(* IEC 61131-3 sources: Mini-Conveyors-Automation/plc, 10 files *)

(* ---- types.st ---- *)
(* =============================================================================
   types.st - Type Definitions
   Mini-Fulfillment Conveyor System

   Enumerations and structures used throughout the PLC program.
   ============================================================================= *)

(* System operating states *)
TYPE E_SystemState :
(
    STOPPED  := 0,   (* System is idle, motor off, safe to interact *)
    STARTING := 1,   (* Pre-run checks in progress *)
    RUNNING  := 2,   (* Normal operation, conveyor moving *)
    FAULT    := 3    (* Fault condition active, motor off, alarm on *)
);
END_TYPE

(* Fault codes *)
TYPE E_FaultCode :
(
    NONE            := 0,   (* No fault *)
    ESTOP           := 1,   (* Emergency stop activated *)
    JAM_INFEED      := 2,   (* Jam detected at infeed photoeye *)
    JAM_DIVERTER    := 3,   (* Jam detected at diverter photoeye *)
    JAM_OUTFEED_B   := 4,   (* Jam detected at outfeed B photoeye *)
    JAM_OUTFEED_C   := 5    (* Jam detected at outfeed C photoeye *)
);
END_TYPE

(* Operating mode *)
TYPE E_OperatingMode :
(
    AUTO   := 0,   (* Automatic mode - full autonomous operation *)
    MANUAL := 1    (* Manual mode - jog only, no auto routing *)
);
END_TYPE

(* Metrics data structure *)
TYPE ST_Metrics :
STRUCT
    diBoxCount       : DINT;    (* Total boxes processed *)
    rAvgCycleTime    : REAL;    (* Average cycle time in seconds *)
    diJamCount       : DINT;    (* Total jam events *)
    rThroughput      : REAL;    (* Current throughput in boxes/hour *)
    rRunningTime     : REAL;    (* Total running time in seconds *)
    rFaultTime       : REAL;    (* Total fault/downtime in seconds *)
    rLastCycleTime   : REAL;    (* Most recent box cycle time *)
    rCycleTimeSum    : REAL;    (* Sum of all cycle times for averaging *)
END_STRUCT
END_TYPE

(* Jam detection status per photoeye *)
TYPE ST_JamStatus :
STRUCT
    bBlocked         : BOOL;    (* Photoeye currently blocked *)
    bJamDetected     : BOOL;    (* Jam threshold exceeded *)
    tBlockedDuration : TIME;    (* How long PE has been blocked *)
END_STRUCT
END_TYPE

(* ---- global_vars.st ---- *)
(* =============================================================================
   global_vars.st - Global Variables (Global Variable List)
   Mini-Fulfillment Conveyor System

   Shared variables used across program blocks and for HMI binding.
   ============================================================================= *)

VAR_GLOBAL
    (* =========================================================================
       SYSTEM STATE
       ========================================================================= *)
    eSystemState    : E_SystemState := STOPPED;    (* Current system state *)
    eOperatingMode  : E_OperatingMode := AUTO;     (* Current operating mode *)
    eFaultCode      : E_FaultCode := NONE;         (* Active fault code *)
    sFaultMessage   : STRING(80) := '';             (* Active fault description *)

    (* =========================================================================
       SAFETY FLAGS
       ========================================================================= *)
    bSafeToRun      : BOOL := FALSE;   (* TRUE when all safety checks pass *)
    bFaultActive    : BOOL := FALSE;   (* TRUE when any fault is active *)
    bEStopLatched   : BOOL := FALSE;   (* TRUE when E-Stop has been activated, requires clear *)
    bJamDetected    : BOOL := FALSE;   (* TRUE when any photoeye jam is detected *)

    (* =========================================================================
       CONTROL FLAGS
       ========================================================================= *)
    bMotorRunCmd    : BOOL := FALSE;   (* Motor run command from state machine *)
    bRejectNext     : BOOL := FALSE;   (* TRUE = next box routes to Station C *)
    diBoxCounter    : DINT := 0;       (* Running box count for routing pattern *)

    (* =========================================================================
       JAM DETECTION STATUS
       ========================================================================= *)
    stJamInfeed     : ST_JamStatus;    (* Jam status for infeed PE *)
    stJamDiverter   : ST_JamStatus;    (* Jam status for diverter PE *)
    stJamOutfeedB   : ST_JamStatus;    (* Jam status for outfeed B PE *)
    stJamOutfeedC   : ST_JamStatus;    (* Jam status for outfeed C PE *)

    (* =========================================================================
       METRICS
       ========================================================================= *)
    stMetrics       : ST_Metrics;      (* Aggregated metrics structure *)

    (* =========================================================================
       HMI INTERFACE - Commands (HMI -> PLC)
       ========================================================================= *)
    bHMI_Start      : BOOL := FALSE;   (* Start command from HMI *)
    bHMI_Stop       : BOOL := FALSE;   (* Stop command from HMI *)
    bHMI_FaultClear : BOOL := FALSE;   (* Fault clear command from HMI *)
    bHMI_JogFwd     : BOOL := FALSE;   (* Jog forward command from HMI (manual mode) *)

    (* =========================================================================
       HMI INTERFACE - Parameters (HMI -> PLC)
       ========================================================================= *)
    rJamTimeoutSec  : REAL := 4.0;     (* Jam detection timeout in seconds (adjustable) *)
    rConveyorSpeed  : REAL := 1.0;     (* Conveyor speed setpoint 0.0 to 1.0 (1.0 = full speed) *)

    (* =========================================================================
       HMI INTERFACE - Status (PLC -> HMI)
       ========================================================================= *)
    iHMI_State      : INT := 0;        (* System state as INT for HMI display *)
    sHMI_FaultMsg   : STRING(80) := '';(* Fault message for HMI display *)
    rHMI_BoxCount   : DINT := 0;       (* Box count for HMI display *)
    rHMI_AvgCycleTime : REAL := 0.0;   (* Avg cycle time for HMI display *)
    rHMI_JamCount   : DINT := 0;       (* Jam count for HMI display *)
    rHMI_Throughput : REAL := 0.0;     (* Throughput for HMI display *)

    (* =========================================================================
       TIMING
       ========================================================================= *)
    tCycleStartTime : TIME := T#0S;    (* Timestamp when current box entered infeed *)
    bCycleActive    : BOOL := FALSE;   (* TRUE when a box is being tracked through the system *)
END_VAR

(* ---- io_mapping.st ---- *)
(* =============================================================================
   io_mapping.st - I/O Address Mapping (Global Variable List)
   Mini-Fulfillment Conveyor System

   Maps physical I/O addresses to symbolic names.
   This GVL is the ONLY place where physical addresses appear.
   All other program blocks reference these symbolic names.
   ============================================================================= *)

VAR_GLOBAL
    (* =========================================================================
       DIGITAL INPUTS
       ========================================================================= *)

    (* Operator panel *)
    bStartPB       AT %IX0.0 : BOOL;   (* Start pushbutton - NO, TRUE on press *)
    bStopPB        AT %IX0.1 : BOOL;   (* Stop pushbutton - NC, FALSE on press *)
    bEStop         AT %IX0.2 : BOOL;   (* E-Stop - NC, FALSE when activated *)
    bModeSelector  AT %IX0.3 : BOOL;   (* Mode switch - FALSE=Auto, TRUE=Manual *)

    (* Photoeyes - TRUE when blocked by a box *)
    bInfeedPE      AT %IX1.0 : BOOL;   (* Infeed photoeye at Station A *)
    bDiverterPE    AT %IX1.1 : BOOL;   (* Diverter photoeye at routing point *)
    bOutfeedBPE    AT %IX1.2 : BOOL;   (* Outfeed B photoeye at Station B (accept) *)
    bOutfeedCPE    AT %IX1.3 : BOOL;   (* Outfeed C photoeye at Station C (reject) *)

    (* =========================================================================
       DIGITAL OUTPUTS
       ========================================================================= *)

    bConveyorMotor     AT %QX0.0 : BOOL;   (* Main conveyor belt motor *)
    bDiverterActuator  AT %QX0.1 : BOOL;   (* Diverter gate solenoid - FALSE=StationB, TRUE=StationC *)
    bAlarmBuzzer       AT %QX0.2 : BOOL;   (* Fault alarm buzzer *)
    bStatusGreen       AT %QX0.3 : BOOL;   (* Green status light - RUNNING *)
    bStatusRed         AT %QX0.4 : BOOL;   (* Red status light - FAULT *)
END_VAR

(* ---- fb_conveyor.st ---- *)
(* =============================================================================
   FB_Conveyor - Conveyor Motor Control Function Block
   Mini-Fulfillment Conveyor System

   Controls the main conveyor belt motor based on system state and mode.
   Provides speed reference output for potential variable-speed drive.
   ============================================================================= *)

FUNCTION_BLOCK FB_Conveyor
VAR_INPUT
    bRunCommand     : BOOL;         (* Motor run command from state machine *)
    bJogCommand     : BOOL;         (* Jog command from manual mode *)
    bManualMode     : BOOL;         (* TRUE when in manual mode *)
    rSpeedSetpoint  : REAL := 1.0;  (* Speed setpoint 0.0 to 1.0 *)
END_VAR

VAR_OUTPUT
    bMotorOutput    : BOOL;         (* Final motor on/off command *)
    rSpeedRef       : REAL;         (* Speed reference output (0.0 to 1.0) *)
    bMotorRunning   : BOOL;         (* Feedback: motor is currently running *)
END_VAR

VAR
    rJogSpeed       : REAL := 0.3;  (* Jog speed as fraction of full speed *)
END_VAR

(* --- Determine motor state --- *)
IF bManualMode THEN
    (* Manual mode: motor runs only while jog is held *)
    bMotorOutput := bJogCommand;
    IF bJogCommand THEN
        rSpeedRef := rJogSpeed;     (* Reduced speed for jogging *)
    ELSE
        rSpeedRef := 0.0;
    END_IF
ELSE
    (* Auto mode: motor runs continuously when commanded *)
    bMotorOutput := bRunCommand;
    IF bRunCommand THEN
        rSpeedRef := rSpeedSetpoint;
    ELSE
        rSpeedRef := 0.0;
    END_IF
END_IF

(* --- Motor running feedback --- *)
bMotorRunning := bMotorOutput;

(* ---- fb_diverter.st ---- *)
(* =============================================================================
   FB_Diverter - Accept/Reject Routing Function Block
   Mini-Fulfillment Conveyor System

   Controls the diverter gate to route boxes to Station B (accept) or
   Station C (reject). Uses a pattern-based accept/reject decision for
   deterministic testing (every 3rd box is rejected).

   Diverter safe state: de-energized (FALSE) = Station B (accept path).
   ============================================================================= *)

FUNCTION_BLOCK FB_Diverter
VAR_INPUT
    bInfeedPE       : BOOL;         (* Infeed photoeye - box arrived *)
    bDiverterPE     : BOOL;         (* Diverter photoeye - box at decision point *)
    bSystemRunning  : BOOL;         (* TRUE when system is RUNNING in AUTO mode *)
    bAutoMode       : BOOL;         (* TRUE when in auto mode *)
END_VAR

VAR_OUTPUT
    bDiverterOutput : BOOL := FALSE;    (* Diverter actuator command *)
    bRejectActive   : BOOL := FALSE;    (* TRUE when current box is being rejected *)
    diBoxCounter    : DINT := 0;        (* Running box counter for pattern *)
END_VAR

VAR
    bInfeedPrev     : BOOL := FALSE;    (* Previous scan infeed PE for edge detection *)
    bDiverterPrev   : BOOL := FALSE;    (* Previous scan diverter PE for edge detection *)
    bInfeedRising   : BOOL := FALSE;    (* Infeed PE rising edge *)
    bDiverterRising : BOOL := FALSE;    (* Diverter PE rising edge *)
    bDiverterFalling : BOOL := FALSE;   (* Diverter PE falling edge *)
    bRejectNext     : BOOL := FALSE;    (* Flag: next box should be rejected *)
    bDiverterLocked : BOOL := FALSE;    (* Diverter position locked while box is at gate *)
END_VAR

(* Only process routing in auto mode while running *)
IF bSystemRunning AND bAutoMode THEN

    (* --- Edge Detection --- *)
    bInfeedRising := bInfeedPE AND NOT bInfeedPrev;
    bDiverterRising := bDiverterPE AND NOT bDiverterPrev;
    bDiverterFalling := NOT bDiverterPE AND bDiverterPrev;

    (* --- Box Arrival at Infeed: determine accept/reject --- *)
    IF bInfeedRising THEN
        diBoxCounter := diBoxCounter + 1;

        (* Pattern: every 3rd box is rejected *)
        IF (diBoxCounter MOD 3) = 0 THEN
            bRejectNext := TRUE;
        ELSE
            bRejectNext := FALSE;
        END_IF
    END_IF

    (* --- Box Reaches Diverter: actuate if reject --- *)
    IF bDiverterRising THEN
        bDiverterLocked := TRUE;
        IF bRejectNext THEN
            bDiverterOutput := TRUE;    (* Energize = route to Station C *)
            bRejectActive := TRUE;
        ELSE
            bDiverterOutput := FALSE;   (* De-energized = route to Station B *)
            bRejectActive := FALSE;
        END_IF
    END_IF

    (* --- Box Clears Diverter: return to safe position --- *)
    IF bDiverterFalling AND bDiverterLocked THEN
        bDiverterOutput := FALSE;       (* Return to safe position *)
        bDiverterLocked := FALSE;
        bRejectActive := FALSE;
        bRejectNext := FALSE;           (* Clear flag for next box *)
    END_IF

ELSE
    (* Not running or in manual mode: diverter in safe position *)
    bDiverterOutput := FALSE;
    bRejectActive := FALSE;
    bDiverterLocked := FALSE;
END_IF

(* --- Update previous states --- *)
bInfeedPrev := bInfeedPE;
bDiverterPrev := bDiverterPE;

(* ---- fb_jam_detection.st ---- *)
(* =============================================================================
   FB_JamDetection - Jam Detection and Fault Handling Function Block
   Mini-Fulfillment Conveyor System

   Monitors all photoeyes for jam conditions. A jam is detected when any
   photoeye remains blocked for longer than the configurable timeout.
   Identifies the jam location and provides fault clear logic.
   ============================================================================= *)

FUNCTION_BLOCK FB_JamDetection
VAR_INPUT
    bInfeedPE       : BOOL;         (* Infeed photoeye state *)
    bDiverterPE     : BOOL;         (* Diverter photoeye state *)
    bOutfeedBPE     : BOOL;         (* Outfeed B photoeye state *)
    bOutfeedCPE     : BOOL;         (* Outfeed C photoeye state *)
    bSystemRunning  : BOOL;         (* TRUE when system is in RUNNING state *)
    bFaultClear     : BOOL;         (* Fault clear command *)
    rJamTimeoutSec  : REAL := 4.0;  (* Jam timeout in seconds (configurable from HMI) *)
END_VAR

VAR_OUTPUT
    bJamDetected    : BOOL := FALSE;    (* TRUE when any jam is active *)
    eFaultCode      : E_FaultCode;      (* Fault code identifying jam location *)
    sFaultMessage   : STRING(80);       (* Fault description *)
    stInfeedJam     : ST_JamStatus;     (* Infeed PE jam status *)
    stDiverterJam   : ST_JamStatus;     (* Diverter PE jam status *)
    stOutfeedBJam   : ST_JamStatus;     (* Outfeed B PE jam status *)
    stOutfeedCJam   : ST_JamStatus;     (* Outfeed C PE jam status *)
END_VAR

VAR
    tonInfeed       : TON;      (* Jam timer for infeed PE *)
    tonDiverter     : TON;      (* Jam timer for diverter PE *)
    tonOutfeedB     : TON;      (* Jam timer for outfeed B PE *)
    tonOutfeedC     : TON;      (* Jam timer for outfeed C PE *)
    tJamTimeout     : TIME;     (* Jam timeout as TIME value *)
    bFaultClearPrev : BOOL := FALSE;    (* Previous scan fault clear *)
    bFaultClearRising : BOOL := FALSE;  (* Rising edge of fault clear *)
    bJamLatched     : BOOL := FALSE;    (* Jam fault is latched until cleared *)
END_VAR

(* --- Convert timeout parameter --- *)
tJamTimeout := REAL_TO_TIME(rJamTimeoutSec * 1000.0);  (* seconds to milliseconds *)

(* --- Edge detection on fault clear --- *)
bFaultClearRising := bFaultClear AND NOT bFaultClearPrev;
bFaultClearPrev := bFaultClear;

(* --- Only monitor for jams while system is running or jam is latched --- *)
IF bSystemRunning OR bJamLatched THEN

    (* === Infeed Photoeye Jam Timer === *)
    tonInfeed(IN := bInfeedPE AND bSystemRunning, PT := tJamTimeout);
    stInfeedJam.bBlocked := bInfeedPE;
    stInfeedJam.tBlockedDuration := tonInfeed.ET;

    IF tonInfeed.Q AND NOT bJamLatched THEN
        stInfeedJam.bJamDetected := TRUE;
        bJamLatched := TRUE;
        eFaultCode := E_FaultCode.JAM_INFEED;
        sFaultMessage := 'JAM DETECTED AT INFEED (Station A)';
    END_IF

    (* === Diverter Photoeye Jam Timer === *)
    tonDiverter(IN := bDiverterPE AND bSystemRunning, PT := tJamTimeout);
    stDiverterJam.bBlocked := bDiverterPE;
    stDiverterJam.tBlockedDuration := tonDiverter.ET;

    IF tonDiverter.Q AND NOT bJamLatched THEN
        stDiverterJam.bJamDetected := TRUE;
        bJamLatched := TRUE;
        eFaultCode := E_FaultCode.JAM_DIVERTER;
        sFaultMessage := 'JAM DETECTED AT DIVERTER';
    END_IF

    (* === Outfeed B Photoeye Jam Timer === *)
    tonOutfeedB(IN := bOutfeedBPE AND bSystemRunning, PT := tJamTimeout);
    stOutfeedBJam.bBlocked := bOutfeedBPE;
    stOutfeedBJam.tBlockedDuration := tonOutfeedB.ET;

    IF tonOutfeedB.Q AND NOT bJamLatched THEN
        stOutfeedBJam.bJamDetected := TRUE;
        bJamLatched := TRUE;
        eFaultCode := E_FaultCode.JAM_OUTFEED_B;
        sFaultMessage := 'JAM DETECTED AT OUTFEED B (Station B)';
    END_IF

    (* === Outfeed C Photoeye Jam Timer === *)
    tonOutfeedC(IN := bOutfeedCPE AND bSystemRunning, PT := tJamTimeout);
    stOutfeedCJam.bBlocked := bOutfeedCPE;
    stOutfeedCJam.tBlockedDuration := tonOutfeedC.ET;

    IF tonOutfeedC.Q AND NOT bJamLatched THEN
        stOutfeedCJam.bJamDetected := TRUE;
        bJamLatched := TRUE;
        eFaultCode := E_FaultCode.JAM_OUTFEED_C;
        sFaultMessage := 'JAM DETECTED AT OUTFEED C (Station C)';
    END_IF

ELSE
    (* System not running and no latched jam: reset all timers *)
    tonInfeed(IN := FALSE);
    tonDiverter(IN := FALSE);
    tonOutfeedB(IN := FALSE);
    tonOutfeedC(IN := FALSE);
END_IF

(* --- Jam Fault Clear Logic --- *)
(* Clear jam when: operator presses fault clear AND the jammed PE is no longer blocked *)
IF bJamLatched AND bFaultClearRising THEN
    CASE eFaultCode OF
        E_FaultCode.JAM_INFEED:
            IF NOT bInfeedPE THEN
                bJamLatched := FALSE;
                stInfeedJam.bJamDetected := FALSE;
                eFaultCode := E_FaultCode.NONE;
                sFaultMessage := '';
            END_IF

        E_FaultCode.JAM_DIVERTER:
            IF NOT bDiverterPE THEN
                bJamLatched := FALSE;
                stDiverterJam.bJamDetected := FALSE;
                eFaultCode := E_FaultCode.NONE;
                sFaultMessage := '';
            END_IF

        E_FaultCode.JAM_OUTFEED_B:
            IF NOT bOutfeedBPE THEN
                bJamLatched := FALSE;
                stOutfeedBJam.bJamDetected := FALSE;
                eFaultCode := E_FaultCode.NONE;
                sFaultMessage := '';
            END_IF

        E_FaultCode.JAM_OUTFEED_C:
            IF NOT bOutfeedCPE THEN
                bJamLatched := FALSE;
                stOutfeedCJam.bJamDetected := FALSE;
                eFaultCode := E_FaultCode.NONE;
                sFaultMessage := '';
            END_IF
    END_CASE
END_IF

(* --- Aggregate jam status --- *)
bJamDetected := bJamLatched;

(* ---- fb_manual_mode.st ---- *)
(* =============================================================================
   FB_ManualMode - Manual / Jog Control Function Block
   Mini-Fulfillment Conveyor System

   Provides manual jog control for the conveyor. In manual mode, the
   conveyor runs only while the jog button is held, at reduced speed.
   Safety interlocks remain active. No automatic routing occurs.
   ============================================================================= *)

FUNCTION_BLOCK FB_ManualMode
VAR_INPUT
    bManualMode     : BOOL;         (* TRUE when mode selector = Manual *)
    bJogFwdPB       : BOOL;         (* Jog forward pushbutton (or HMI button) *)
    bSystemRunning  : BOOL;         (* TRUE when system state = RUNNING *)
    bSafeToRun      : BOOL;         (* Safety permissive from FB_Safety *)
END_VAR

VAR_OUTPUT
    bMotorJogCmd    : BOOL := FALSE;    (* Motor jog command *)
    bJogActive      : BOOL := FALSE;    (* TRUE while jogging *)
END_VAR

VAR
    (* No internal variables needed for basic jog *)
END_VAR

(* --- Jog Logic --- *)
(* Jog is allowed only when:
   1. System is in RUNNING state
   2. Mode selector is set to Manual
   3. Safety permissive is TRUE
   4. Jog button is held
*)

IF bManualMode AND bSystemRunning AND bSafeToRun THEN
    IF bJogFwdPB THEN
        bMotorJogCmd := TRUE;
        bJogActive := TRUE;
    ELSE
        bMotorJogCmd := FALSE;
        bJogActive := FALSE;
    END_IF
ELSE
    bMotorJogCmd := FALSE;
    bJogActive := FALSE;
END_IF

(* ---- fb_metrics.st ---- *)
(* =============================================================================
   FB_Metrics - Metrics Tracking Function Block
   Mini-Fulfillment Conveyor System

   Tracks operational metrics:
   - Box count (total processed)
   - Cycle time (infeed to outfeed, running average)
   - Jam count
   - Throughput (boxes per hour)
   - Running time vs fault/downtime
   ============================================================================= *)

FUNCTION_BLOCK FB_Metrics
VAR_INPUT
    bInfeedPE       : BOOL;         (* Infeed photoeye *)
    bOutfeedBPE     : BOOL;         (* Outfeed B photoeye *)
    bOutfeedCPE     : BOOL;         (* Outfeed C photoeye *)
    bSystemRunning  : BOOL;         (* TRUE when state = RUNNING *)
    bFaultState     : BOOL;         (* TRUE when state = FAULT *)
    bJamEvent       : BOOL;         (* Rising edge triggers jam count increment *)
    tScanTime       : TIME := T#10MS;   (* PLC scan time for time accumulation *)
END_VAR

VAR_OUTPUT
    stMetrics       : ST_Metrics;   (* Output metrics structure *)
END_VAR

VAR
    (* Edge detection *)
    bInfeedPrev     : BOOL := FALSE;
    bOutfeedBPrev   : BOOL := FALSE;
    bOutfeedCPrev   : BOOL := FALSE;
    bJamEventPrev   : BOOL := FALSE;

    (* Cycle time measurement *)
    bCycleActive    : BOOL := FALSE;    (* A box is being tracked *)
    tCycleTimer     : TON;              (* Timer for current box cycle *)
    rCurrentCycle   : REAL := 0.0;      (* Current cycle time in seconds *)

    (* Time accumulation *)
    tRunTimer       : TON;              (* Accumulates running time *)
    tFaultTimer     : TON;              (* Accumulates fault time *)
    rScanTimeSec    : REAL;             (* Scan time converted to seconds *)

    (* Edge signals *)
    bInfeedRising   : BOOL;
    bOutfeedBRising : BOOL;
    bOutfeedCRising : BOOL;
    bJamRising      : BOOL;
END_VAR

(* --- Compute scan time in seconds --- *)
rScanTimeSec := TIME_TO_REAL(tScanTime) / 1000.0;

(* --- Edge Detection --- *)
bInfeedRising := bInfeedPE AND NOT bInfeedPrev;
bOutfeedBRising := bOutfeedBPE AND NOT bOutfeedBPrev;
bOutfeedCRising := bOutfeedCPE AND NOT bOutfeedCPrev;
bJamRising := bJamEvent AND NOT bJamEventPrev;

(* =========================================================================
   BOX CYCLE TIME TRACKING
   ========================================================================= *)

(* Start cycle timer when box arrives at infeed *)
IF bInfeedRising AND NOT bCycleActive THEN
    bCycleActive := TRUE;
    tCycleTimer(IN := FALSE);   (* Reset timer *)
END_IF

(* Run cycle timer while tracking a box *)
IF bCycleActive THEN
    tCycleTimer(IN := TRUE, PT := T#300S);  (* Max 300s cycle, should never reach *)
END_IF

(* Complete cycle when box reaches either outfeed *)
IF bCycleActive AND (bOutfeedBRising OR bOutfeedCRising) THEN
    (* Record cycle time *)
    rCurrentCycle := TIME_TO_REAL(tCycleTimer.ET) / 1000.0;  (* Convert to seconds *)
    stMetrics.rLastCycleTime := rCurrentCycle;

    (* Increment box count *)
    stMetrics.diBoxCount := stMetrics.diBoxCount + 1;

    (* Update running average *)
    stMetrics.rCycleTimeSum := stMetrics.rCycleTimeSum + rCurrentCycle;
    IF stMetrics.diBoxCount > 0 THEN
        stMetrics.rAvgCycleTime := stMetrics.rCycleTimeSum / DINT_TO_REAL(stMetrics.diBoxCount);
    END_IF

    (* Reset cycle tracking *)
    bCycleActive := FALSE;
    tCycleTimer(IN := FALSE);
END_IF

(* =========================================================================
   JAM COUNT
   ========================================================================= *)
IF bJamRising THEN
    stMetrics.diJamCount := stMetrics.diJamCount + 1;
END_IF

(* =========================================================================
   RUNNING TIME AND FAULT TIME ACCUMULATION
   ========================================================================= *)

(* Accumulate running time using scan-by-scan addition *)
IF bSystemRunning THEN
    stMetrics.rRunningTime := stMetrics.rRunningTime + rScanTimeSec;
END_IF

IF bFaultState THEN
    stMetrics.rFaultTime := stMetrics.rFaultTime + rScanTimeSec;
END_IF

(* =========================================================================
   THROUGHPUT CALCULATION
   ========================================================================= *)

(* Throughput = boxes per hour *)
IF stMetrics.rRunningTime > 1.0 THEN  (* Avoid division by zero, wait at least 1 second *)
    stMetrics.rThroughput := DINT_TO_REAL(stMetrics.diBoxCount) / (stMetrics.rRunningTime / 3600.0);
ELSE
    stMetrics.rThroughput := 0.0;
END_IF

(* =========================================================================
   UPDATE PREVIOUS STATES
   ========================================================================= *)
bInfeedPrev := bInfeedPE;
bOutfeedBPrev := bOutfeedBPE;
bOutfeedCPrev := bOutfeedCPE;
bJamEventPrev := bJamEvent;

(* ---- fb_safety.st ---- *)
(* =============================================================================
   FB_Safety - Safety and Interlock Function Block
   Mini-Fulfillment Conveyor System

   Monitors E-Stop, evaluates safety interlocks, and provides a safe-to-run
   permissive signal. E-Stop is latching: once activated, it requires both
   the E-Stop to be reset (circuit closed) AND a Fault Clear command.
   ============================================================================= *)

FUNCTION_BLOCK FB_Safety
VAR_INPUT
    bEStop          : BOOL;     (* E-Stop input - NC circuit: TRUE = healthy, FALSE = activated *)
    bStopPB         : BOOL;     (* Stop pushbutton - NC: TRUE = not pressed, FALSE = pressed *)
    bStartPB        : BOOL;     (* Start pushbutton - NO: TRUE = pressed *)
    bFaultClear     : BOOL;     (* Fault clear command (pushbutton or HMI) *)
    bJamActive      : BOOL;     (* Jam fault from FB_JamDetection *)
END_VAR

VAR_OUTPUT
    bSafeToRun      : BOOL;     (* TRUE when all safety conditions met for running *)
    bFaultActive    : BOOL;     (* TRUE when any fault is active *)
    bEStopLatched   : BOOL;     (* TRUE when E-Stop has been activated and not yet cleared *)
    bStartCmd       : BOOL;     (* Rising edge of start command, qualified by safety *)
    bStopCmd        : BOOL;     (* Stop command detected *)
    eFaultCode      : E_FaultCode;  (* Active fault code *)
    sFaultMessage   : STRING(80);   (* Fault description text *)
END_VAR

VAR
    bEStopPrev      : BOOL := TRUE;     (* Previous scan E-Stop state for edge detection *)
    bStartPrev      : BOOL := FALSE;    (* Previous scan start PB for rising edge *)
    bStopPrev       : BOOL := TRUE;     (* Previous scan stop PB for falling edge *)
    bFaultClearPrev : BOOL := FALSE;    (* Previous scan fault clear for rising edge *)
    bStartRisingEdge : BOOL := FALSE;   (* One-shot start command *)
    bFaultClearRising : BOOL := FALSE;  (* One-shot fault clear *)
END_VAR

(* --- Edge Detection --- *)
bStartRisingEdge := bStartPB AND NOT bStartPrev;
bFaultClearRising := bFaultClear AND NOT bFaultClearPrev;

(* --- E-Stop Latching Logic --- *)
(* E-Stop is NC: TRUE = healthy. When it goes FALSE, latch the fault. *)
IF NOT bEStop THEN
    bEStopLatched := TRUE;
    eFaultCode := E_FaultCode.ESTOP;
    sFaultMessage := 'EMERGENCY STOP ACTIVATED';
END_IF

(* --- E-Stop Latch Clear --- *)
(* Clear only when: E-Stop circuit is healthy again AND operator requests clear *)
IF bEStopLatched AND bFaultClearRising AND bEStop THEN
    bEStopLatched := FALSE;
    (* Only clear fault code if no other faults active *)
    IF NOT bJamActive THEN
        eFaultCode := E_FaultCode.NONE;
        sFaultMessage := '';
    END_IF
END_IF

(* --- Aggregate Fault Status --- *)
bFaultActive := bEStopLatched OR bJamActive;

(* --- Update fault code/message for jam (if E-Stop not the cause) --- *)
IF bJamActive AND NOT bEStopLatched THEN
    (* Fault code for jam is set by FB_JamDetection via global vars *)
    (* We just ensure bFaultActive stays TRUE *)
    ;
END_IF

(* --- Safe-to-Run Permissive --- *)
(* All conditions must be TRUE for the system to be allowed to run *)
bSafeToRun := bEStop              (* E-Stop circuit healthy *)
          AND NOT bEStopLatched   (* No latched E-Stop fault *)
          AND NOT bJamActive      (* No active jam *)
          AND bStopPB;            (* Stop PB not pressed (NC = TRUE when not pressed) *)

(* --- Start Command (qualified) --- *)
(* Only issue start if safety permits *)
bStartCmd := bStartRisingEdge AND bSafeToRun;

(* --- Stop Command --- *)
(* Stop detected on falling edge of NC stop button (TRUE -> FALSE) *)
bStopCmd := bStopPrev AND NOT bStopPB;

(* --- Update previous states for next scan --- *)
bEStopPrev := bEStop;
bStartPrev := bStartPB;
bStopPrev := bStopPB;
bFaultClearPrev := bFaultClear;

(* ---- prg_main.st ---- *)
(* =============================================================================
   PRG_Main - Main Program (State Machine Orchestrator)
   Mini-Fulfillment Conveyor System

   Central state machine that coordinates all function blocks.
   Called every scan cycle by MainTask (10 ms).
   ============================================================================= *)

PROGRAM PRG_Main
VAR
    (* Function block instances *)
    fbSafety        : FB_Safety;
    fbConveyor      : FB_Conveyor;
    fbJamDetection  : FB_JamDetection;
    fbDiverter      : FB_Diverter;
    fbManualMode    : FB_ManualMode;
    fbMetrics       : FB_Metrics;

    (* Internal state *)
    tonStartDelay   : TON;              (* 1-second startup delay timer *)
    bStartDelayDone : BOOL := FALSE;    (* Startup delay completed *)
    bBlinkToggle    : BOOL := FALSE;    (* For blinking status lights *)
    tonBlink        : TON;              (* Blink timer - 500ms period *)
    tBlinkTime      : TIME := T#500MS;  (* Blink half-period *)
END_VAR

(* =========================================================================
   1. READ OPERATING MODE
   ========================================================================= *)
IF IO_Mapping.bModeSelector THEN
    GVL.eOperatingMode := E_OperatingMode.MANUAL;
ELSE
    GVL.eOperatingMode := E_OperatingMode.AUTO;
END_IF

(* =========================================================================
   2. EXECUTE SAFETY BLOCK
   ========================================================================= *)
fbSafety(
    bEStop      := IO_Mapping.bEStop,
    bStopPB     := IO_Mapping.bStopPB,
    bStartPB    := IO_Mapping.bStartPB OR GVL.bHMI_Start,
    bFaultClear := GVL.bHMI_FaultClear,
    bJamActive  := GVL.bJamDetected
);

(* Update global safety flags *)
GVL.bSafeToRun    := fbSafety.bSafeToRun;
GVL.bFaultActive  := fbSafety.bFaultActive;
GVL.bEStopLatched := fbSafety.bEStopLatched;

(* =========================================================================
   2b. EXECUTE JAM DETECTION BLOCK
   ========================================================================= *)
fbJamDetection(
    bInfeedPE       := IO_Mapping.bInfeedPE,
    bDiverterPE     := IO_Mapping.bDiverterPE,
    bOutfeedBPE     := IO_Mapping.bOutfeedBPE,
    bOutfeedCPE     := IO_Mapping.bOutfeedCPE,
    bSystemRunning  := (GVL.eSystemState = E_SystemState.RUNNING),
    bFaultClear     := GVL.bHMI_FaultClear,
    rJamTimeoutSec  := GVL.rJamTimeoutSec
);

(* Update global jam status *)
GVL.bJamDetected  := fbJamDetection.bJamDetected;
GVL.stJamInfeed   := fbJamDetection.stInfeedJam;
GVL.stJamDiverter := fbJamDetection.stDiverterJam;
GVL.stJamOutfeedB := fbJamDetection.stOutfeedBJam;
GVL.stJamOutfeedC := fbJamDetection.stOutfeedCJam;

(* Use jam fault info if jam is active, otherwise use safety fault info *)
IF fbJamDetection.bJamDetected THEN
    GVL.eFaultCode    := fbJamDetection.eFaultCode;
    GVL.sFaultMessage := fbJamDetection.sFaultMessage;
ELSE
    GVL.eFaultCode    := fbSafety.eFaultCode;
    GVL.sFaultMessage := fbSafety.sFaultMessage;
END_IF

(* =========================================================================
   2c. EXECUTE CONVEYOR BLOCK
   ========================================================================= *)
fbConveyor(
    bRunCommand     := GVL.bMotorRunCmd,
    bJogCommand     := GVL.bHMI_JogFwd,
    bManualMode     := (GVL.eOperatingMode = E_OperatingMode.MANUAL),
    rSpeedSetpoint  := GVL.rConveyorSpeed
);

(* =========================================================================
   3. STATE MACHINE
   ========================================================================= *)
CASE GVL.eSystemState OF

    (* ----- STOPPED ----- *)
    E_SystemState.STOPPED:
        (* Outputs in safe state *)
        GVL.bMotorRunCmd := FALSE;
        IO_Mapping.bDiverterActuator := FALSE;
        IO_Mapping.bAlarmBuzzer := FALSE;
        IO_Mapping.bStatusGreen := FALSE;
        IO_Mapping.bStatusRed := FALSE;

        (* Transition: Start command received and safe to run *)
        IF fbSafety.bStartCmd THEN
            GVL.eSystemState := E_SystemState.STARTING;
            tonStartDelay(IN := FALSE);  (* Reset timer *)
            bStartDelayDone := FALSE;
        END_IF

    (* ----- STARTING ----- *)
    E_SystemState.STARTING:
        GVL.bMotorRunCmd := FALSE;
        IO_Mapping.bDiverterActuator := FALSE;
        IO_Mapping.bAlarmBuzzer := FALSE;

        (* Blink green light during startup *)
        IO_Mapping.bStatusGreen := bBlinkToggle;
        IO_Mapping.bStatusRed := FALSE;

        (* 1-second startup delay *)
        tonStartDelay(IN := TRUE, PT := T#1S);
        IF tonStartDelay.Q THEN
            bStartDelayDone := TRUE;
        END_IF

        (* Check for faults during startup *)
        IF GVL.bFaultActive THEN
            GVL.eSystemState := E_SystemState.FAULT;
        ELSIF bStartDelayDone AND GVL.bSafeToRun THEN
            (* All pre-run checks passed *)
            GVL.eSystemState := E_SystemState.RUNNING;
        END_IF

    (* ----- RUNNING ----- *)
    E_SystemState.RUNNING:
        IO_Mapping.bStatusGreen := TRUE;
        IO_Mapping.bStatusRed := FALSE;
        IO_Mapping.bAlarmBuzzer := FALSE;

        (* Motor control depends on mode *)
        IF GVL.eOperatingMode = E_OperatingMode.AUTO THEN
            GVL.bMotorRunCmd := TRUE;
        ELSE
            (* Manual mode: motor controlled by FB_ManualMode *)
            ; (* FB_ManualMode sets bMotorRunCmd *)
        END_IF

        (* Transition to FAULT *)
        IF GVL.bFaultActive THEN
            GVL.eSystemState := E_SystemState.FAULT;
            GVL.bMotorRunCmd := FALSE;
        END_IF

        (* Transition to STOPPED on stop command *)
        IF fbSafety.bStopCmd OR GVL.bHMI_Stop THEN
            GVL.eSystemState := E_SystemState.STOPPED;
            GVL.bMotorRunCmd := FALSE;
        END_IF

    (* ----- FAULT ----- *)
    E_SystemState.FAULT:
        GVL.bMotorRunCmd := FALSE;
        IO_Mapping.bDiverterActuator := FALSE;  (* Safe position *)
        IO_Mapping.bStatusGreen := FALSE;
        IO_Mapping.bStatusRed := bBlinkToggle;  (* Blink red *)
        IO_Mapping.bAlarmBuzzer := TRUE;

        (* Transition to STOPPED when fault is cleared *)
        IF NOT GVL.bFaultActive THEN
            GVL.eSystemState := E_SystemState.STOPPED;
            IO_Mapping.bAlarmBuzzer := FALSE;
        END_IF

END_CASE

(* =========================================================================
   4. BLINK TIMER (used for status light blinking)
   ========================================================================= *)
tonBlink(IN := NOT tonBlink.Q, PT := tBlinkTime);
IF tonBlink.Q THEN
    bBlinkToggle := NOT bBlinkToggle;
END_IF

(* =========================================================================
   5. APPLY MOTOR OUTPUT (safety gating)
   ========================================================================= *)
(* Final motor output: run command AND all safety conditions *)
IO_Mapping.bConveyorMotor := GVL.bMotorRunCmd
                         AND IO_Mapping.bEStop
                         AND NOT GVL.bEStopLatched
                         AND IO_Mapping.bStopPB;

(* =========================================================================
   6. UPDATE HMI TAGS
   ========================================================================= *)
GVL.iHMI_State      := TO_INT(GVL.eSystemState);
GVL.sHMI_FaultMsg   := GVL.sFaultMessage;
GVL.rHMI_BoxCount   := GVL.stMetrics.diBoxCount;
GVL.rHMI_AvgCycleTime := GVL.stMetrics.rAvgCycleTime;
GVL.rHMI_JamCount   := GVL.stMetrics.diJamCount;
GVL.rHMI_Throughput := GVL.stMetrics.rThroughput;

(* Reset one-shot HMI commands after processing *)
GVL.bHMI_Start := FALSE;
GVL.bHMI_Stop := FALSE;
GVL.bHMI_FaultClear := FALSE;
